{attribute 'pack_mode' := '1'}
TYPE ST_Chiller_Writes :
STRUCT
	controlOut : ST_Control;
	valueOut : ST_Value0;
END_STRUCT
END_TYPE

(* stored: Version 1.1.0.1
   DUT ST_Chiller_Writes: Id {6161c4da-d70f-4889-85b4-afa73b59614b} *)
